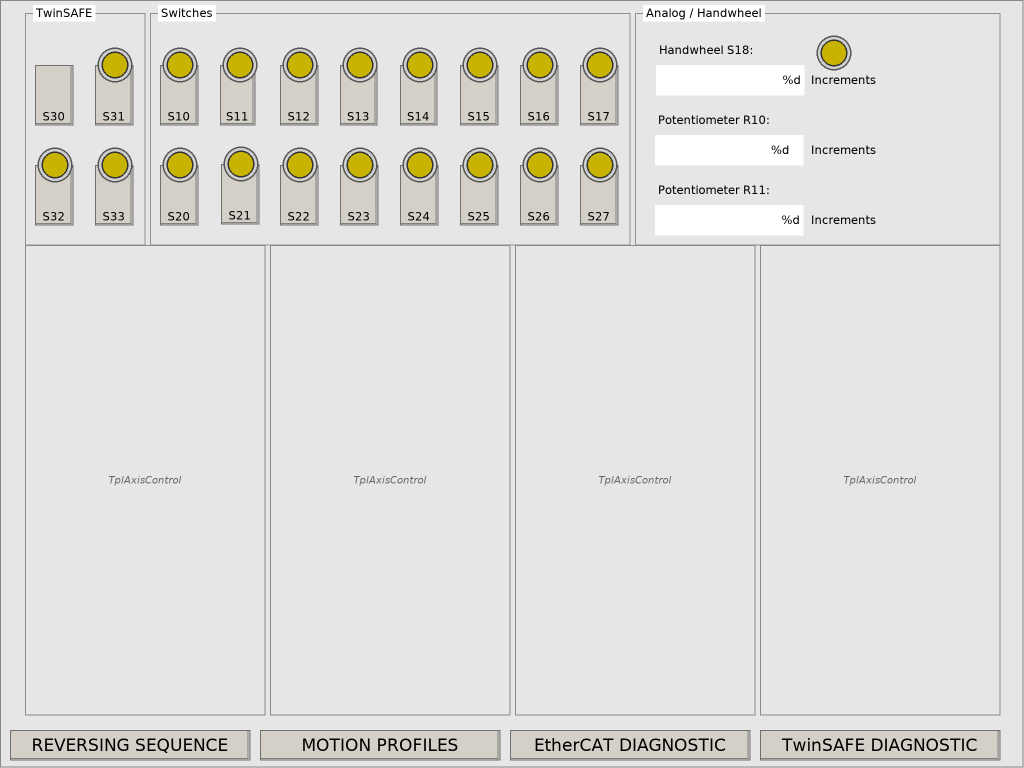
VISUALIZATION HmiStartPage  // 1024x768
    Rectangle (0,0 1024x768)
    Button (760,730 240x30), "TwinSAFE DIAGNOSTIC"
        OnMouseClick: change screen: HmiTwinSAFEDiagnostic
    Button (510,730 240x30), "EtherCAT DIAGNOSTIC"
        OnMouseClick: change screen: HmiEtherCatDiagnostic
    GroupBox (25,5 120x240), "TwinSAFE"
        Button (10,60 38x60), "S30", colour toggle: NOT TwinSAFE.fbSafeConnectionEL1904_1_Group1.bChannel1 and NOT TwinSAFE.fbSafeConnectionEL1904_1_Group1.bChannel2
            toggle bSwitchS31
        Button (70,60 38x60), "S31", colour toggle: bSwitchS31
            toggle bSwitchS31
        Lamp1 (70,40 40x40), variable: bLedH31, style: Lamp-Lamp1-Yellow
        Button (70,160 38x60), "S33", colour toggle: NOT TwinSAFE.fbSafeConnectionEL1904_2_Group1.bChannel3 and TwinSAFE.fbSafeConnectionEL1904_2_Group1.bChannel4
            toggle bSwitchS31
        Lamp1 (70,140 40x40), variable: bLedH33, style: Lamp-Lamp1-Yellow
        Button (10,160 38x60), "S32", colour toggle: NOT TwinSAFE.fbSafeConnectionEL1904_2_Group1.bChannel1 and NOT TwinSAFE.fbSafeConnectionEL1904_2_Group1.bChannel2
            toggle bSwitchS31
        Lamp1 (10,140 40x40), variable: bLedH32, style: Lamp-Lamp1-Yellow
    GroupBox (150,5 480x240), "Switches"
        Button (10,60 38x60), "S10", colour toggle: bSwitchS10
            toggle bSwitchS10
        Lamp1 (10,40 40x40), variable: bLedH10, style: Lamp-Lamp1-Yellow
        Button (70,60 35x60), "S11", colour toggle: bSwitchS11
            toggle bSwitchS11
        Lamp1 (70,40 40x40), variable: bLedH11, style: Lamp-Lamp1-Yellow
        Button (130,60 38x60), "S12", colour toggle: bSwitchS12
            toggle bSwitchS12
        Lamp1 (130,40 40x40), variable: bLedH12, style: Lamp-Lamp1-Yellow
        Button (190,60 37x60), "S13", colour toggle: bSwitchS13
            toggle bSwitchS13
        Lamp1 (190,40 40x40), variable: bLedH13, style: Lamp-Lamp1-Yellow
        Button (250,60 37x60), "S14", colour toggle: bSwitchS14
            toggle bSwitchS14
        Lamp1 (250,40 40x40), variable: bLedH14, style: Lamp-Lamp1-Yellow
        Button (310,60 38x60), "S15", colour toggle: bSwitchS15
            toggle bSwitchS15
        Lamp1 (310,40 40x40), variable: bLedH15, style: Lamp-Lamp1-Yellow
        Button (370,60 38x60), "S16", colour toggle: bSwitchS16
            toggle bSwitchS16
        Lamp1 (370,40 40x40), variable: bLedH16, style: Lamp-Lamp1-Yellow
        Button (430,60 38x60), "S17", colour toggle: bSwitchS17
            toggle bSwitchS17
        Lamp1 (430,40 40x40), variable: bLedH17, style: Lamp-Lamp1-Yellow
        Button (10,160 38x60), "S20", colour toggle: bSwitchS20
            toggle bSwitchS20
        Lamp1 (10,140 40x40), variable: bLedH20, style: Lamp-Lamp1-Yellow
        Button (71,159 38x60), "S21", colour toggle: bSwitchS21
            toggle bSwitchS21
        Lamp1 (71,139 40x40), variable: bLedH21, style: Lamp-Lamp1-Yellow
        Button (130,160 38x60), "S22", colour toggle: bSwitchS22
            toggle bSwitchS22
        Lamp1 (130,140 40x40), variable: bLedH22, style: Lamp-Lamp1-Yellow
        Button (190,160 38x60), "S23", colour toggle: bSwitchS23
            toggle bSwitchS23
        Lamp1 (190,140 40x40), variable: bLedH23, style: Lamp-Lamp1-Yellow
        Button (250,160 38x60), "S24", colour toggle: bSwitchS24
            toggle bSwitchS24
        Lamp1 (250,140 40x40), variable: bLedH24, style: Lamp-Lamp1-Yellow
        Button (310,160 38x60), "S25", colour toggle: bSwitchS25
            toggle bSwitchS25
        Lamp1 (310,140 40x40), variable: bLedH25, style: Lamp-Lamp1-Yellow
        Button (370,160 38x60), "S26", colour toggle: nAX5203DigitalInputs.2
            toggle nAX5203DigitalInputs.2
        Lamp1 (370,140 40x40), variable: bLedH26, style: Lamp-Lamp1-Yellow
        Button (430,160 38x60), "S27", colour toggle: nAX5203DigitalInputs.3
            toggle nAX5203DigitalInputs.3
        Lamp1 (430,140 40x40), variable: nAX5203DigitalOutputs.7, style: Lamp-Lamp1-Yellow
    GroupBox (635,5 365x240), "Analog / Handwheel"
        Rectangle (20,200 148x30), "%d", text variable: aOsAnalogInR11[0]
            OnMouseClick: write the text variable via VisuDialogs.Numpad, min 0, max 32767
        Label (173,200 118x30), "Increments"
        Label (20,170 197x30), "Potentiometer R11:"
        Rectangle (20,130 148x30), "%d", text variable: nAnalogInR10
            OnMouseClick: write the text variable via VisuDialogs.Numpad, min 0, max 32767
        Label (173,130 121x30), "Increments"
        Label (20,100 216x30), "Potentiometer R10:"
        Lamp1 (179,28 40x40), variable: bHandwheelSwitchS28, style: Lamp-Lamp1-Yellow
        Rectangle (21,60 148x30), "%d", text variable: nHandwheelCounter
            OnMouseClick: write the text variable via VisuDialogs.Numpad
        Label (173,60 133x30), "Increments"
        Label (21,30 216x30), "Handwheel S18:"
    Frame (25,245 240x470)
        shows TplAxisControl(sAxisDescription := Axis1.sAxisDescription, fAbsolutePositon := stAxis1.NcToPlc.ActPos, fModuloPositon := stAxis1.NcToPlc.ModuloActPos, bError := Axis1.bAxisErr, nErrorId := Axis1.nAxisErrId, bReset := Axis1.bReset, bPowerStatus := Axis1.fbAxis.bPowerStatus, bReferenceCam := bStepperReferenceCam, fMoveAbsPosition := Axis1.fMoveAbsPosition, fMoveAbsVelocity := Axis1.fMoveAbsVelocity, bStartMoveAbs := Axis1.bStartMoveAbs, bMoveAbsBusy := Axis1.bMoveAbsBusy, bMoveAbsDone := Axis1.bMoveAbsDone, bStop := Axis1.bStop, bStopBusy := Axis1.bStopAxisBusy, bStopDone := Axis1.bStopAxisDone, bAxisCoupled := Axis1.bAxisCoupled, bTestChangeTargetPosAxis := Axis1.bTestChangeTargetPos)
    Frame (270,245 240x470)
        shows TplAxisControl(sAxisDescription := Axis2.sAxisDescription, fAbsolutePositon := stAxis2.NcToPlc.ActPos, fModuloPositon := stAxis2.NcToPlc.ModuloActPos, bError := Axis2.bAxisErr, nErrorId := Axis2.nAxisErrId, bReset := Axis2.bReset, bPowerStatus := Axis2.fbAxis.bPowerStatus, bReferenceCam := bAxis2ReferenceCamEL7, fMoveAbsPosition := Axis2.fMoveAbsPosition, fMoveAbsVelocity := Axis2.fMoveAbsVelocity, bStartMoveAbs := Axis2.bStartMoveAbs, bMoveAbsBusy := Axis2.bMoveAbsBusy, bMoveAbsDone := Axis2.bMoveAbsDone, bStop := Axis2.bStop, bStopBusy := Axis2.bStopAxisBusy, bStopDone := Axis2.bStopAxisDone, bAxisCoupled := Axis2.bAxisCoupled, bTestChangeTargetPosAxis := Axis2.bTestChangeTargetPos)
    Frame (515,245 240x470)
        shows TplAxisControl(sAxisDescription := Axis3.sAxisDescription, fAbsolutePositon := stAxis3.NcToPlc.ActPos, fModuloPositon := stAxis3.NcToPlc.ModuloActPos, bError := Axis3.bAxisErr, nErrorId := Axis3.nAxisErrId, bReset := Axis3.bReset, bPowerStatus := Axis3.fbAxis.bPowerStatus, bReferenceCam := AxisGeneral.bAxis3ReferenceCam, fMoveAbsPosition := Axis3.fMoveAbsPosition, fMoveAbsVelocity := Axis3.fMoveAbsVelocity, bStartMoveAbs := Axis3.bStartMoveAbs, bMoveAbsBusy := Axis3.bMoveAbsBusy, bMoveAbsDone := Axis3.bMoveAbsDone, bStop := Axis3.bStop, bStopBusy := Axis3.bStopAxisBusy, bStopDone := Axis3.bStopAxisDone, bAxisCoupled := Axis3.bAxisCoupled, bTestChangeTargetPosAxis := Axis3.bTestChangeTargetPos)
    Frame (760,245 240x470)
        shows TplAxisControl(sAxisDescription := Axis4.sAxisDescription, fAbsolutePositon := stAxis4.NcToPlc.ActPos, fModuloPositon := stAxis4.NcToPlc.ModuloActPos, bError := Axis4.bAxisErr, nErrorId := Axis4.nAxisErrId, bReset := Axis4.bReset, bPowerStatus := Axis4.fbAxis.bPowerStatus, bReferenceCam := AxisGeneral.bAxis4ReferenceCam, fMoveAbsPosition := Axis4.fMoveAbsPosition, fMoveAbsVelocity := Axis4.fMoveAbsVelocity, bStartMoveAbs := Axis4.bStartMoveAbs, bMoveAbsBusy := Axis4.bMoveAbsBusy, bMoveAbsDone := Axis4.bMoveAbsDone, bStop := Axis4.bStop, bStopBusy := Axis4.bStopAxisBusy, bStopDone := Axis4.bStopAxisDone, bAxisCoupled := Axis4.bAxisCoupled, bTestChangeTargetPosAxis := Axis4.bTestChangeTargetPos)
    Button (10,730 240x30), "REVERSING SEQUENCE"
        OnMouseClick: change screen: HmiAxisReversingSequence
    Button (260,730 240x30), "MOTION PROFILES"
        OnMouseClick: change screen: MotionProfiles
END_VISUALIZATION

(* stored: Version 1.1.0.1
   Visu HmiStartPage: Id {81da00b4-351b-4bea-beba-4843bfdabd99} *)
